PROGRAM DerotatorControl
VAR_INPUT
	// enable the derotator
	enable:		BOOL;
	// reset an error
	reset:		BOOL;
	// decrease derotator angle
	left:		BOOL;
	// increase derotator angle
	right:		BOOL;
	// set the absolute position
	position:	LREAL;
	// derotator velocity
	Velocity:	LREAL := 10.0;
	// move to given position
	MoveAxis: 	BOOL;
	// calibrate the axis
	HomeAxis:	BOOL;
	// tracking flag
	Tracking:	BOOL;
	// stop the Axis
	StopAxis:	BOOL;
	// diagnostic error code reset
	bSoEReset: 			BOOL;
END_VAR
VAR_OUTPUT
	// error flag
	Error:				BOOL;
	// nc error id
	ErrorID:			UDINT;
	// actual position of the derotator
	actual_position:	LREAL;
	// calibrated flag
	Calibrated:			BOOL;
	// axis ready flag
	Ready:				BOOL;
	// position to move the axis to
	slewtime: 			LREAL;
END_VAR
VAR
	// trigger for the torque error
	TorqueError:		TON := (PT := T#3S);
	// axis function block
	DerotatorAxis:		FB_Axis2;
	
	DerotatorEvent:		FB_EventLog;
	// torque warning event
	TorqueWarning:		FB_EventLog;
	// torque calibration event
	CalibrationEvent:	FB_EventLog;
	// diagnostic low-level event
	DerotatorDiagnosticEvent: FB_EventLog;
	// percentage of the derotator torque
	derotator_torque:	REAL;
	// read slewtime
	ReadParameter:		MC_ReadParameter;
	fbSoEReset: 		FB_SoEReset;
	DiagnosticError:	BOOL;
END_VAR
VAR CONSTANT
	// current position of the calibration cam. Apply an offset here if necessary
	calibration_position:	LREAL := 438.4623; // calibration in positive direction (was 460.0)
END_VAR

(*
Selection 6
Homing in Endlage:

https://infosys.beckhoff.com/index.php?content=../content/1031/ax5000_usermanual/html/ax5000_homing_hardware_end_position.htm&id=12221
NC-Interface:
PlcToNc-Achsinterface, Bit 8 namens AcceptBlockedDriveSignal im nDeCtrlDWord

SPS-Interface:
TcNc-Lib, siehe SPS-Funktion AxisSetAcceptBlockedDriveSignal in der TwinCAT  PLC Library: NC.
*)

position := LIMIT(-50, position, 400);

IF enable AND NOT DerotatorAxis.Calibrated THEN
	HomeAxis := TRUE;
END_IF

IF DerotatorAxis.Calibrated THEN
	HomeAxis := FALSE;
	Calibrated := DerotatorAxis.Calibrated;
END_IF
	
IF HomeAxis THEN
	position := calibration_position;
END_IF

DeRotatorAxis(
	enable := 			enable,
	Reset := 			Reset,
	MoveAxis :=			MoveAxis,
	HomeAxis :=			HomeAxis,
	StopAxis :=			StopAxis,
	HomingMode :=		MC_ForceCalibration,
	Position := 		position, 
	Velocity :=			Velocity,
	Enable_Positive := 	NOT GVL_Telescope.Derotator_inputs.0,
	Enable_Negative := 	NOT GVL_Telescope.Derotator_inputs.1,
	Jog_Forward := 		right,
	Jog_Backwards := 	left,
	bCalibrationCam :=	GVL_Telescope.Derotator_inputs.0,
	isModuloAxis :=		FALSE,
	Tracking :=			Tracking,
	ActualPosition => 	actual_position,
	Error => 			Error,
	ErrorID => 			ErrorID,
	AxisRef :=			GVL_Telescope.DerotatorAxisRef);
	
IF DeRotatorAxis.MoveDone OR Reset OR Error THEN
	MoveAxis := FALSE;
END_IF

IF DeRotatorAxis.HomeDone OR Reset OR Error THEN
	HomeAxis := FALSE;
END_IF
	
IF DeRotatorAxis.ResetDone THEN
	reset := FALSE;
END_IF

IF DeRotatorAxis.StopDone THEN
	StopAxis := FALSE;
END_IF

DiagnosticError := FALSE;
IF GVL_Telescope.Derotator_diagnostic < 16#D012 AND GVL_Telescope.Derotator_diagnostic > 16#D014 THEN
	DiagnosticError := TRUE;
	ErrorID := GVL_Telescope.Derotator_diagnostic;
	bSoeReset := reset;
END_IF

Ready := DeRotatorAxis.Ready;

ReadParameter(	Axis := GVL_Telescope.DerotatorAxisRef, 
				Enable := DeRotatorAxis.InMotion, 
				ParameterNumber := MC_AxisParameter.AxisRemainingTimeToGo, 
				ReadMode := E_ReadMode.READMODE_CYCLIC);
				
IF ReadParameter.Valid THEN
	slewtime := ReadParameter.Value;
END_IF

IF bSoEReset THEN
	fbSoEReset(
		Axis := GVL_Telescope.DerotatorAxisRef,
		Execute := TRUE,
		Timeout := DEFAULT_ADS_TIMEOUT);
 	IF NOT fbSoEReset.Busy THEN
		fbSoEReset(Axis := GVL_Telescope.DerotatorAxisRef, Execute := FALSE);
		bSoEReset := FALSE;
		Reset := TRUE;
	END_IF
END_IF

derotator_torque := GVL_Telescope.Derotator_torque / 10.0;
// nominal torque is 3%, max is 25%
TorqueError(IN := ABS(derotator_torque) > 20.0);

DerotatorEvent(	
	Trigger := 		Error, 
	Level := 		ADSLOG_MSGTYPE_ERROR,
	FormatString :=	'Derotator Axis Error: %s',
	OnMessage := 	NCError_TO_STRING(ErrorID),
	OffMEssage := 	'OK',
	OffLevel := 	ADSLOG_MSGTYPE_HINT);
	
DerotatorDiagnosticEvent(	
	Trigger := 		DiagnosticError, 
	Level := 		ADSLOG_MSGTYPE_ERROR,
	FormatString :=	'Derotator Axis Diagnostic Error: %s',
	OnMessage := 	NCError_TO_STRING(GVL_Telescope.Derotator_diagnostic));
	
TorqueWarning(	
	Trigger := 		TorqueError.Q, 
	Level := 		ADSLOG_MSGTYPE_WARN,
	FormatString :=	'%s',
	OnMessage := 	'Derotator torque is high.');

CalibrationEvent(	
	Trigger := 		Calibrated, 
	Level := 		ADSLOG_MSGTYPE_HINT,
	OnMessage := 	'Derotator is calibrated.');

END_PROGRAM

(* stored: Version 1.1.0.1, ProductVersion 3.1.4026.8
   POU DerotatorControl: Id {75f3d994-c6e1-4455-a5dc-0a32056448e8}, SpecialFunc None *)
